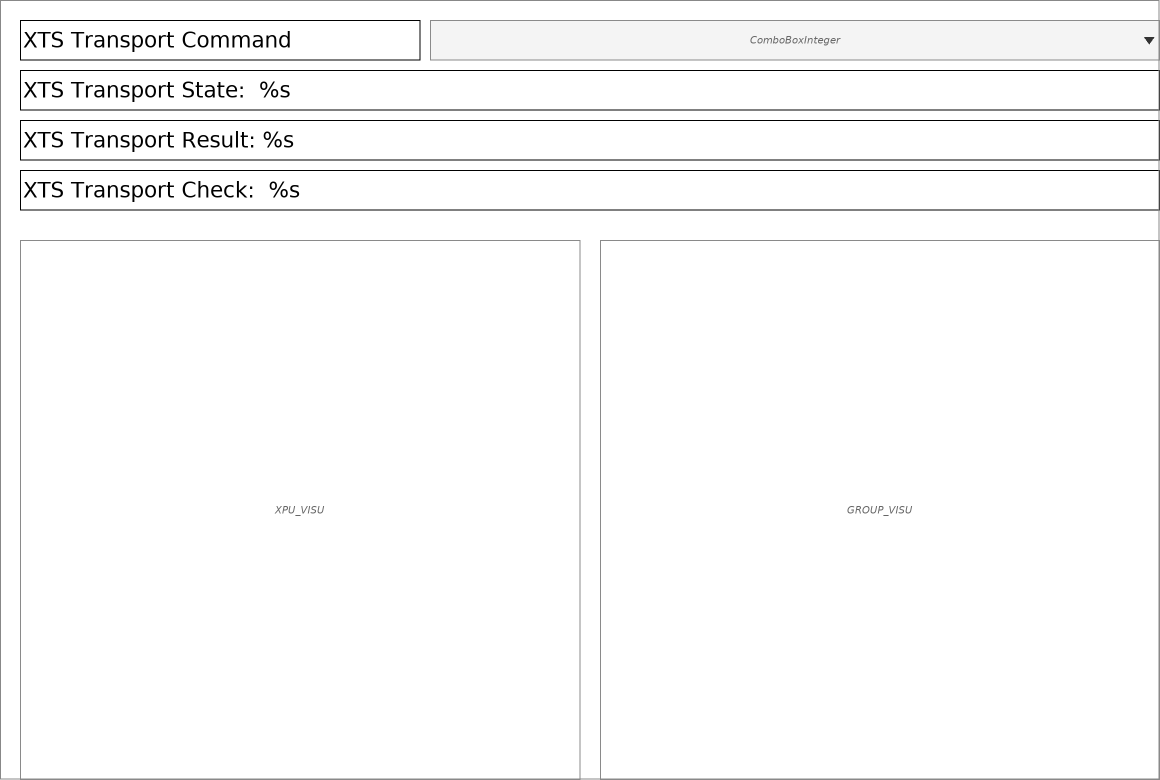
VISUALIZATION XTS_TRANSPORT  // 1160x780
    Rectangle (20,20 400x40), "XTS Transport Command"
    ComboBoxInteger (430,20 730x40), variable: GVL_XTS.XtsTransportCtrl.Cmd, text list: 'TL_E_CTRL_TRANSPORT'
    Frame (20,240 560x540)
        shows XPU_VISU()
    Frame (600,240 560x540)
        shows GROUP_VISU()
    Rectangle (20,70 1140x40), "XTS Transport State: %s", text variable: MAIN.sTransportState
    Rectangle (20,120 1140x40), "XTS Transport Result: %s", text variable: MAIN.sTransportResult
    Rectangle (20,170 1140x40), "XTS Transport Check: %s", text variable: MAIN.sTransportCheck
END_VISUALIZATION

(* stored: Version 1.1.0.1, ProductVersion 3.1.4024.15
   Visu XTS_TRANSPORT: Id {1677eb1f-a145-4dc2-89c6-13c253be66e6} *)
